FUNCTION Convert_UINT_TO_DT : Hresult
VAR_INPUT
	in : UINT;
	out : REFERENCE TO DT;
END_VAR
VAR
	converted : DT;
END_VAR
VAR CONSTANT
	INCOMPATIBLE : HRESULT := 16#9811070E;
END_VAR

converted := UINT_TO_DT(in);

IF (DT_TO_UINT(converted) <> in) THEN
	Convert_UINT_TO_DT := INCOMPATIBLE;
	RETURN;
END_IF

out := converted;

END_FUNCTION

(* stored: Version 1.1.0.1, ProductVersion 3.1.4024.12
   POU Convert_UINT_TO_DT: Id {3c832ee3-4644-4efe-a43c-5d4fa63c9e81}, SpecialFunc None *)
